PROGRAM PRG_00_General
VAR
	sr_Fault: SR;
	FB_Blinker_ServoError: FB_Blinker;
END_VAR

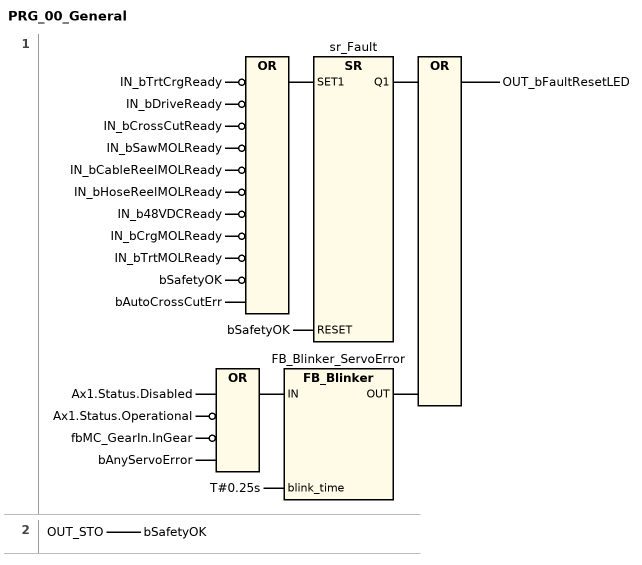
// NETWORK 1
sr_Fault(SET1 := NOT IN_bTrtCrgReady OR NOT IN_bDriveReady OR NOT IN_bCrossCutReady OR NOT IN_bSawMOLReady OR NOT IN_bCableReelMOLReady OR NOT IN_bHoseReelMOLReady OR NOT IN_b48VDCReady OR NOT IN_bCrgMOLReady OR NOT IN_bTrtMOLReady OR NOT bSafetyOK OR bAutoCrossCutErr, RESET := bSafetyOK); // SR
FB_Blinker_ServoError(IN := Ax1.Status.Disabled OR NOT Ax1.Status.Operational OR NOT fbMC_GearIn.InGear OR bAnyServoError, blink_time := T#0.25s); // FB_Blinker
OUT_bFaultResetLED := sr_Fault.Q1 OR FB_Blinker_ServoError.OUT;

// NETWORK 2
bSafetyOK := OUT_STO;

END_PROGRAM

(* stored: Version 1.1.0.1, ProductVersion 3.1.4024.12
   POU PRG_00_General: Id {f29c6036-feae-433d-9645-b299c30f24e8}, SpecialFunc None *)
